RoboDK station: arqui_robot.rdk

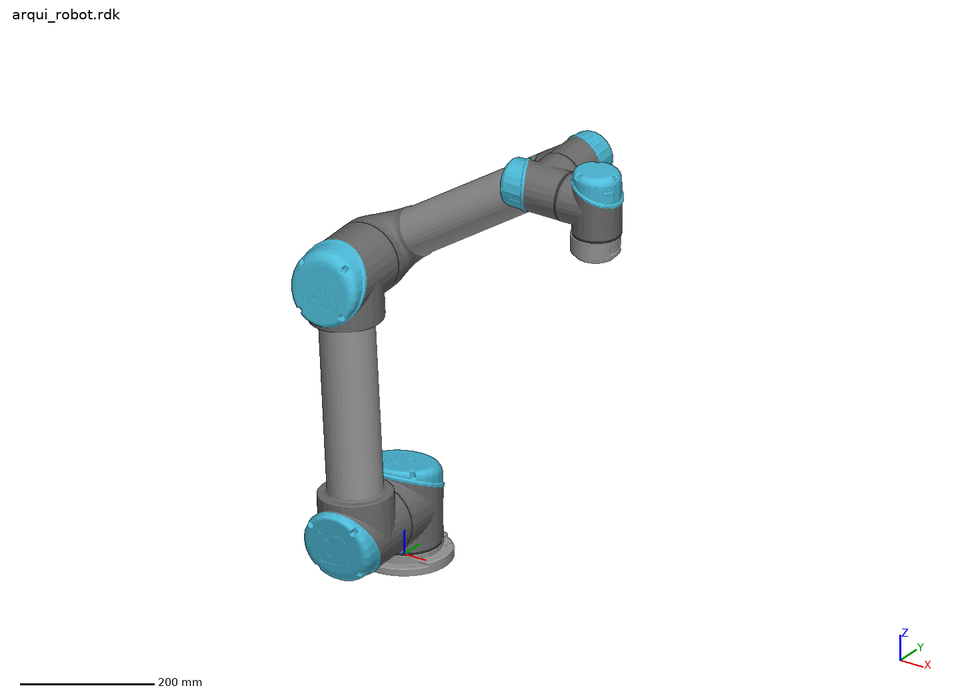
[picture v0: the station drawn from its stored meshes, robots at their saved joint values, targets as dots, program paths as lines]
Station arqui_robot (saved by RoboDK 5.5.1). Poses are relative to the parent item; angles as X-Y-Z fixed-axis rotations.
Station parameters (name, value as stored): FILE_OPENSTATION, C:/Users/pedro/OneDrive - Universidad Técnica Federico Santa María/External-projects/robodk_arqui/rdk_files/arqui_robot.rdk
  - frame UR5 Base at (19.42, 862.3, 631.54) mm
    - robot UR5: 6 axes, payload 5 kg, reach 850 mm, repeatability 0.1 mm, weight 18.4 kg
        modified DH rows (alpha deg, a mm, theta deg, d mm): 0, 0, 0, 89.2; 90, 0, 180, 0; 0, 425, 0, 0; 0, 392.43, 0, 109; -90, 0, 0, 93.65; 90, 0, 180, 82
        joint limits [-360, -360, -360, -360, -360, -360] to [360, 360, 360, 360, 360, 360]; home [0, -90, -90, 0, 90, 0]; saved at [3.852, -86.887, -60.235, -124.132, 90.677, 2.222]
